// SIMATIC S7-200 project (STEP 7-Micro/WIN), CPU 221 REL 01.10

SYMBOL_TABLE USER1
s0               I0.0     // nut nhan khoi dong he thong
s1               I0.1     // nut nhan chay dong co M1 va mo chan
s2               I0.2     // stop
s3               I0.3     // do le nhiet
LC               Q0.0     // la chan mo duoi day thung
BT1              Q0.1     // bang tai 1
H                Q0.2     // den bao he thong hoat dong
END_SYMBOL_TABLE

ORGANIZATION_BLOCK MAIN:OB1
TITLE=PROGRAM COMMENTS
BEGIN
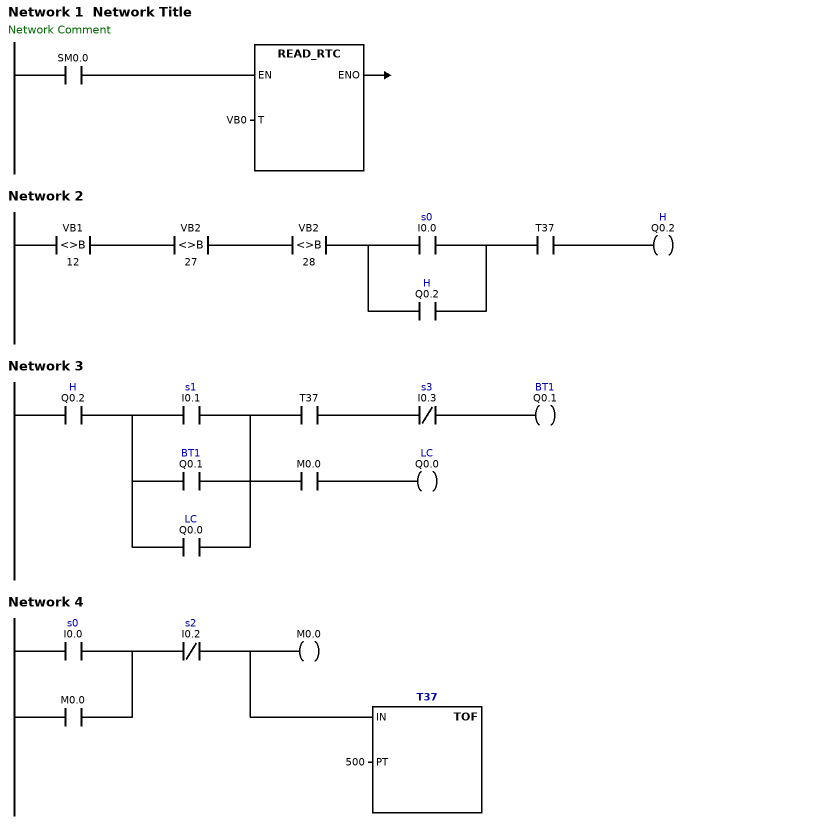
Network 1 // Network Title
// Network Comment
LD     SM0.0
TODR   VB0
Network 2
LDB<>  VB1, 12
AB<>   VB2, 27
AB<>   VB2, 28
LD     s0:I0.0
O      H:Q0.2
ALD
A      T37
=      H:Q0.2
Network 3
LD     H:Q0.2
LD     s1:I0.1
O      BT1:Q0.1
O      LC:Q0.0
ALD
LPS
A      T37
AN     s3:I0.3
=      BT1:Q0.1
LPP
A      M0.0
=      LC:Q0.0
Network 4
LD     s0:I0.0
O      M0.0
AN     s2:I0.2
=      M0.0
TOF    T37, 500
END_ORGANIZATION_BLOCK
